PROGRAM MAIN
VAR
	Position		: LREAL;
	Velocity		: LREAL;
	
	rand			: ARRAY[0..1] OF DRAND;
	i				: INT;
	ton				: TON;
	
	iWriteMe		: DINT := 0;
END_VAR

ton(IN:=NOT ton.Q, PT:=T#1S);
IF ton.Q THEN
	FOR i := 0 TO 1 DO
		rand[i](Seed:=i);
	END_FOR
	
	Position := Position + rand[0].Num;
	Velocity := rand[1].Num * 100;
END_IF

END_PROGRAM

(* stored: Version 1.1.0.1, ProductVersion 3.1.4024.12
   POU MAIN: Id {a902c8b3-6411-414b-8b84-a839e13c6035}, SpecialFunc None *)
